TYPE ST130_PatroneAushebenPos_e :
(
    down_GS,
    up_AS,
    _max
);
END_TYPE

(* stored: Version 1.1.0.1, ProductVersion 3.1.4024.6
   DUT ST130_PatroneAushebenPos_e: Id {f5880163-cbc1-4a1a-81f4-153588247eda} *)
